{attribute 'GeneratedUsingTerminal: EK1122-0000-0018'}
{attribute addProperty BoxType "EK1122-0000-0018"}
{attribute addProperty Id "Beckhoff_APS4xxxsub_EK1100EK1100_AB5A94672A_0001_APS4322_7000_0017APS4322_9345AD93282"}
{attribute addProperty CRC "1934908770"}
{attribute addProperty Size "284"}
TYPE Beckhoff_APS4xxxEK1122_73545D62 EXTENDS EK1122_AB5A9467 :
STRUCT
	{attribute addProperty Name "Beckhoff_APS4xxxsub_EK1100"}
	{attribute addProperty PreviousPort "Beckhoff APS4xxxEK1122 : D"}
	Beckhoff_APS4xxxsub_EK1100 : EK1100_AB5A9467;
	{attribute addProperty Name "A_0001_APS4322_7000_0017"}
	{attribute addProperty PreviousPort "Beckhoff APS4xxxsub EK1100 : C"}
	A_0001_APS4322_7000_0017 : APS4322_9345AD93;
END_STRUCT
END_TYPE

(* stored: Version 1.2.0.0, ProductVersion 3.1.4024.9
   DUT Beckhoff_APS4xxxEK1122_73545D62: Id {638b57a9-4110-42f7-8dc4-9eadc102ef6f} *)
